{attribute 'qualified_only'}
VAR_GLOBAL
	sysLog : FB_SysLog;
	auditLog : FB_AuditLog;
END_VAR

(* stored: Version 1.1.0.1
   GVL GVL_FCSLTracing: Id {e4360a75-728d-417b-8b2a-c33f9f75dce4} *)
